INTERFACE I_StringBuilder EXTENDS __SYSTEM.IQueryInterface

METHOD Append : I_StringBuilder
VAR_INPUT
	sText : STRING;
END_VAR
END_METHOD

METHOD Clear : I_StringBuilder
VAR_INPUT
END_VAR
END_METHOD

METHOD ToString : STRING
VAR_INPUT
END_VAR
END_METHOD

END_INTERFACE

(* stored: Version 1.1.0.1, ProductVersion 3.1.4024.12
   Itf I_StringBuilder: Id {2fd0ddb0-5ffd-403c-92a5-7dcdf27733e3}
   Method Append: Id {f510b285-34c4-4542-a396-e0a2e25db2d1}
   Method Clear: Id {85c7c393-6c1f-4aa1-a068-6ced829f413a}
   Method ToString: Id {266dde48-8af4-4476-99b0-29a8ee80b4ba} *)
